Fanuc KAREL source: kt00154.KL

-- PROVISIONAL review KL for V940-1; original PC SHA256 23b829cb3bb6874c4bc70d6ac1f696c2cd26cac18f76a4b39e3399115401fbc8
-- Incomplete behavior may be omitted. Consult companion uncertainty JSON. Do not deploy.
PROGRAM KT00154
%NOLOCKGROUP
VAR
  I2 : INTEGER
  OUT : REAL
-- UNRESOLVED_DECL H1 type=002017
BEGIN
  -- V9_ZERO_TABLE_METADATA_HINT layout=0001; no indexed target words; source/name/runtime held
  -- UNRESOLVED_PC offsets 5-19; opcodes 2E,22,9D,33,B4
  -- UNRESOLVED_PC offsets 24-35; opcodes 2E,23
  -- UNRESOLVED_PC offsets 40-63; opcodes 22,9D,33,B3,21,55,64,23
  -- UNRESOLVED_PC offsets 68-72; opcodes 7F
END KT00154
